(* IEC 61131-3 sources: IEC61131-3-CDSV3/PCRE2/src, 11 files *)

(* ---- eCompileOptions.dut ---- *)
(*#-#-#-#-#-#-#-#-#-#---Declaration---#-#-#-#-#-#-#-#-#-#-#-#-#*)

// PCRE2 compile options.
// These can be combined using bitwise OR operations.
// See also: https://pcre2project.github.io/pcre2/doc/html/pcre2_compile.html
{attribute 'qualified_only'}
TYPE eCompileOptions :
(
	PCRE2_ALLOW_EMPTY_CLASS := 16#00000001,
    PCRE2_ALT_BSUX := 16#00000002,
    PCRE2_ALT_CIRCUMFLEX := 16#00200000,
    PCRE2_ALT_VERBNAMES := 16#00400000,
    PCRE2_ANCHORED := 16#80000000,
    PCRE2_AUTO_CALLOUT := 16#00000004,
    PCRE2_CASELESS := 16#00000008,
    PCRE2_DOLLAR_ENDONLY := 16#00000010,
    PCRE2_DOTALL := 16#00000020,
    PCRE2_DUPNAMES := 16#00000040,
    PCRE2_ENDANCHORED := 16#20000000,
    PCRE2_EXTENDED := 16#00000080,
    PCRE2_EXTENDED_MORE := 16#01000000,
    PCRE2_FIRSTLINE := 16#00000100,
    PCRE2_LITERAL := 16#02000000,
    PCRE2_MATCH_INVALID_UTF := 16#04000000,
    PCRE2_MATCH_UNSET_BACKREF := 16#00000200,
    PCRE2_MULTILINE := 16#00000400,
    PCRE2_NEVER_BACKSLASH_C := 16#00100000,
    PCRE2_NEVER_UCP := 16#00000800,
    PCRE2_NEVER_UTF := 16#00001000,
    PCRE2_NO_AUTO_CAPTURE := 16#00002000,
    PCRE2_NO_AUTO_POSSESS := 16#00004000,
    PCRE2_NO_DOTSTAR_ANCHOR := 16#00008000,
    PCRE2_NO_START_OPTIMIZE := 16#00010000,
    PCRE2_NO_UTF_CHECK := 16#40000000,
    PCRE2_UCP := 16#00020000,
    PCRE2_UNGREEDY := 16#00040000,
    PCRE2_USE_OFFSET_LIMIT := 16#00800000,
    PCRE2_UTF := 16#00080000
) UDINT;
END_TYPE

(* ---- eMatchOptions.dut ---- *)
(*#-#-#-#-#-#-#-#-#-#---Declaration---#-#-#-#-#-#-#-#-#-#-#-#-#*)

// PCRE2 match options.
// These can be combined using bitwise OR operations.
// See also: https://pcre2project.github.io/pcre2/doc/html/pcre2_match.html
{attribute 'qualified_only'}
TYPE eMatchOptions :
(
	PCRE2_NOTBOL := 16#00000001,
    PCRE2_NOTEOL := 16#00000002,
    PCRE2_NOTEMPTY := 16#00000004,
    PCRE2_NOTEMPTY_ATSTART := 16#00000008,
    PCRE2_PARTIAL_SOFT := 16#00000010,
    PCRE2_PARTIAL_HARD := 16#00000020,
    PCRE2_SUBSTITUTE_GLOBAL := 16#00000100, // pcre2_substitute() only
    PCRE2_SUBSTITUTE_EXTENDED := 16#00000200, // pcre2_substitute() only
    PCRE2_SUBSTITUTE_UNSET_EMPTY := 16#00000400, // pcre2_substitute() only
    PCRE2_SUBSTITUTE_UNKNOWN_UNSET := 16#00000800, // pcre2_substitute() only
    PCRE2_SUBSTITUTE_OVERFLOW_LENGTH := 16#00001000, // pcre2_substitute() only
    PCRE2_NO_JIT := 16#00002000,
    PCRE2_COPY_MATCHED_SUBJECT := 16#00004000,
    PCRE2_SUBSTITUTE_LITERAL := 16#00008000, // pcre2_substitute() only
    PCRE2_SUBSTITUTE_MATCHED := 16#00010000, // pcre2_substitute() only
    PCRE2_SUBSTITUTE_REPLACEMENT_ONLY := 16#00020000 // pcre2_substitute() only
) UDINT;
END_TYPE

(* ---- FuCompilePCRE.pou ---- *)
(*#-#-#-#-#-#-#-#-#-#---Declaration---#-#-#-#-#-#-#-#-#-#-#-#-#*)

// Compiles the given pattern into a PCRE compiled pattern.
// Before use, the pattern must be compiled first.
// After use, the compiled pattern MUST be freed.
// The return value is a pointer to the compiled pattern and
// should be given to the other functions as input "re".
// If compilation fails, the return value is 0.
{attribute 'qualified_only'}
FUNCTION FuCompilePCRE : __XWORD
VAR_INPUT
    psPattern: POINTER TO STRING(1);    // The pattern to compile - for technical reasons, this is STRING(1), although any string length is supported
    udiLength: UDINT;                   // The length of the string
    udiOptions: UDINT;                  // Any compile options to be passed to pcre2_compile() (see eCompileOptions, these can be combined with OR)
END_VAR
(*#-#-#-#-#-#-#-#-#-#---Implementation---#-#-#-#-#-#-#-#-#-#-#-#-#*)

IF psPattern = 0 THEN
    RETURN;
END_IF

FuCompilePCRE := FuCompilePCRE_cext(psPattern, udiLength, udiOptions);

(* ---- FuFreeMatchPCRE.pou ---- *)
(*#-#-#-#-#-#-#-#-#-#---Declaration---#-#-#-#-#-#-#-#-#-#-#-#-#*)

// Releases the match block from FuMatchPCRE.
// To prevent memory leaks, you need to free match blocks after use.
{attribute 'qualified_only'}
FUNCTION FuFreeMatchPCRE
VAR_INPUT
    mb: __XWORD;    // Pointer to the match block from FuMatchPCRE
END_VAR
(*#-#-#-#-#-#-#-#-#-#---Implementation---#-#-#-#-#-#-#-#-#-#-#-#-#*)

IF mb = 0 THEN
    RETURN;
END_IF

FuFreeMatchPCRE_cext(mb);

(* ---- FuFreePCRE.pou ---- *)
(*#-#-#-#-#-#-#-#-#-#---Declaration---#-#-#-#-#-#-#-#-#-#-#-#-#*)

// Frees the PCRE compiled pattern.
// This function MUST be called in order to free the underlying resources,
// after you don't need this anymore.
// To prevent memory leaks, you need to free compiled patterns after use.
// You MUST make sure you DO NOT free compiled patterns BEFORE you release any match blocks for the same pattern.
{attribute 'qualified_only'}
FUNCTION FuFreePCRE
VAR_INPUT
    re: __XWORD;    // Pointer to the compiled pattern from FuCompilePCRE
END_VAR
(*#-#-#-#-#-#-#-#-#-#---Implementation---#-#-#-#-#-#-#-#-#-#-#-#-#*)

IF re = 0 THEN
    RETURN;
END_IF

FuFreePCRE_cext(re);

(* ---- FuGetMatchPCRE.pou ---- *)
(*#-#-#-#-#-#-#-#-#-#---Declaration---#-#-#-#-#-#-#-#-#-#-#-#-#*)

// Returns the match substring designated at the index.
// The return value designes whether we have a match at the index and it was successfully fetched.
// This function will also return partial match strings,
// if the match string is not large enough to contain the whole string.
{attribute 'qualified_only'}
FUNCTION FuGetMatchPCRE : BOOL
VAR_INPUT
    mb: __XWORD;                        // Pointer to the match block from FuMatchPCRE
    psSubject: POINTER TO STRING(1);    // The subject to match on - for technical reasons, this is STRING(1), although any string length is supported
    udiSubjectLength: UDINT;            // The length of the subject string
    uiMatchIndex: UINT;                 // The index of the match (maximum one less than the amount of matches)
    psMatch: POINTER TO STRING(1);      // The string to put the match in - for technical reasons, this is STRING(1), although any string length is supported
    udiSize: UDINT;                     // The size (maximum length) of the match string (psMatch)
END_VAR
VAR_OUTPUT
    udiLength: UDINT;                   // The actual length of the match substring
END_VAR
(*#-#-#-#-#-#-#-#-#-#---Implementation---#-#-#-#-#-#-#-#-#-#-#-#-#*)

IF mb = 0 OR_ELSE psSubject = 0 OR_ELSE udiSubjectLength = 0 OR_ELSE psMatch = 0 OR_ELSE udiSize = 0 THEN
    RETURN;
END_IF

FuGetMatchPCRE := FuGetMatchPCRE_cext(mb, psSubject, udiSubjectLength, uiMatchIndex, psMatch, udiSize, udiLength => udiLength);

(* ---- FuGetMatchSubstringLengthPCRE.pou ---- *)
(*#-#-#-#-#-#-#-#-#-#---Declaration---#-#-#-#-#-#-#-#-#-#-#-#-#*)

// Get the match substring length designated at the index.
// The return value designes whether we have a match at the index and it was successfully fetched.
{attribute 'qualified_only'}
FUNCTION FuGetMatchSubstringLengthPCRE : BOOL
VAR_INPUT
    mb: __XWORD;                        // Pointer to the match block from FuMatchPCRE
    uiMatchIndex: UINT;                 // The index of the match (maximum one less than the amount of matches)
END_VAR
VAR_OUTPUT
    udiLength: UDINT;                   // The length of the match substring
END_VAR
(*#-#-#-#-#-#-#-#-#-#---Implementation---#-#-#-#-#-#-#-#-#-#-#-#-#*)

IF mb = 0 THEN
    RETURN;
END_IF

FuGetMatchSubstringLengthPCRE := FuGetMatchSubstringLengthPCRE_cext(mb, uiMatchIndex, udiLength => udiLength);

(* ---- FuGetNamedMatchPCRE.pou ---- *)
(*#-#-#-#-#-#-#-#-#-#---Declaration---#-#-#-#-#-#-#-#-#-#-#-#-#*)

// Returns the match substring designated with the given match name.
// The return value designes whether we have a match with that name and it was successfully fetched.
// This function will also return FALSE, if the match string is not large enough to contain the whole match.
{attribute 'qualified_only'}
FUNCTION FuGetNamedMatchPCRE : BOOL
VAR_INPUT
    mb: __XWORD;                        // Pointer to the match block from FuMatchPCRE
    psSubject: POINTER TO STRING(1);    // The subject to match on - for technical reasons, this is STRING(1), although any string length is supported
    udiSubjectLength: UDINT;            // The length of the subject string
    sMatchName: STRING(255);            // The name of the match
    psMatch: POINTER TO STRING(1);      // The string to put the match in - for technical reasons, this is STRING(1), although any string length is supported
    udiSize: UDINT;                     // The size (maximum length) of the match string (psMatch)
END_VAR
VAR_OUTPUT
    udiLength: UDINT;                   // The actual length of the match substring
END_VAR
(*#-#-#-#-#-#-#-#-#-#---Implementation---#-#-#-#-#-#-#-#-#-#-#-#-#*)

IF mb = 0 OR_ELSE psSubject = 0 OR_ELSE udiSubjectLength = 0 OR_ELSE sMatchName = '' OR_ELSE psMatch = 0 OR_ELSE udiSize = 0 THEN
    RETURN;
END_IF

FuGetNamedMatchPCRE := FuGetNamedMatchPCRE_cext(
    mb,
    psSubject,
    udiSubjectLength,
    sMatchName,
    TO_UDINT(MAX(0, Stu.StrLenA(ADR(sMatchName)))),
    psMatch,
    udiSize,
    udiLength => udiLength
);

(* ---- FuGetNamedMatchSubstringLengthPCRE.pou ---- *)
(*#-#-#-#-#-#-#-#-#-#---Declaration---#-#-#-#-#-#-#-#-#-#-#-#-#*)

// Get the match substring length designated with the given match name.
// The return value designes whether we have a match with that name and it was successfully fetched.
{attribute 'qualified_only'}
FUNCTION FuGetNamedMatchSubstringLengthPCRE : BOOL
VAR_INPUT
    mb: __XWORD;                        // Pointer to the match block from FuMatchPCRE
    sMatchName: STRING(255);            // The name of the match
END_VAR
VAR_OUTPUT
    udiLength: UDINT;                   // The length of the match substring
END_VAR
(*#-#-#-#-#-#-#-#-#-#---Implementation---#-#-#-#-#-#-#-#-#-#-#-#-#*)

IF mb = 0 OR_ELSE sMatchName = '' THEN
    RETURN;
END_IF

FuGetNamedMatchSubstringLengthPCRE := FuGetNamedMatchSubstringLengthPCRE_cext(
    mb,
    sMatchName,
    TO_UDINT(MAX(0, Stu.StrLenA(ADR(sMatchName)))),
    udiLength => udiLength
);

(* ---- FuMatchPCRE.pou ---- *)
(*#-#-#-#-#-#-#-#-#-#---Declaration---#-#-#-#-#-#-#-#-#-#-#-#-#*)

// Matches the subject string against the subject string.
// The return value contains the number of matches. A negative number indicates an error from PCRE2.
//
// The output contains a pointer to the match block, which is needed for FuGetMatchPCRE and FuGetNamedMatchPCRE.
// After use, you need to release the match block using FuFreeMatchPCRE.
// You MUST make sure you DO NOT free compiled patterns BEFORE you release the match block.
{attribute 'qualified_only'}
FUNCTION FuMatchPCRE : INT
VAR_INPUT
    re: __XWORD;                        // Pointer to the compiled pattern from FuCompilePCRE
    psSubject: POINTER TO STRING(1);    // The subject to match on - for technical reasons, this is STRING(1), although any string length is supported
    udiLength: UDINT;                   // The length of the string
    udiOffset: UDINT := 0;              // Offset at the start of the subject string for matching
    udiOptions: UDINT := 0;             // Any valid pcre2_match() options (see eMatchOptions, these can be combined with OR)
END_VAR
VAR_OUTPUT
    mb: __XWORD;                        // The pointer to the match block
END_VAR
(*#-#-#-#-#-#-#-#-#-#---Implementation---#-#-#-#-#-#-#-#-#-#-#-#-#*)

IF re = 0 OR_ELSE psSubject = 0 THEN
    RETURN;
END_IF

FuMatchPCRE := FuMatchPCRE_cext(re, psSubject, udiLength, udiOffset, udiOptions, mb => mb);

(* ---- FuSimpleMatchPCRE.pou ---- *)
(*#-#-#-#-#-#-#-#-#-#---Declaration---#-#-#-#-#-#-#-#-#-#-#-#-#*)

// Simply checks whether the PCRE compiled pattern matches the string.
{attribute 'qualified_only'}
FUNCTION FuSimpleMatchPCRE : BOOL
VAR_INPUT
    re: __XWORD;                        // Pointer to the compiled pattern from FuCompilePCRE
    psSubject: POINTER TO STRING(1);    // The subject to match on - for technical reasons, this is STRING(1), although any string length is supported
    udiLength: UDINT;                   // The length of the string
    udiOffset: UDINT := 0;              // Offset at the start of the subject string for matching
    udiOptions: UDINT := 0;             // Any valid pcre2_match() options (see eMatchOptions, these can be combined with OR)
END_VAR
(*#-#-#-#-#-#-#-#-#-#---Implementation---#-#-#-#-#-#-#-#-#-#-#-#-#*)

IF re = 0 OR_ELSE psSubject = 0 THEN
    RETURN;
END_IF

FuSimpleMatchPCRE := FuSimpleMatchPCRE_cext(re, psSubject, udiLength, udiOffset, udiOptions);
